Staubli VAL3: feedbackStatus.pgx

public program feedbackStatus(num x_nOutConnFlag)
begin

  // update connection status on port 11002 (feedback server)

  gotoxy(scMonitor, 0,1)
  // 11 characteres: gotoxy(12,1) to insert status
  put(scMonitor, "Port 11002:")
  gotoxy(scMonitor, 12,1)
  switch x_nOutConnFlag
    case -1
      put(scMonitor, "connection lost")
    break
    case 0
      put(scMonitor, "not connected")
    break
    case 1
      put(scMonitor, "connected")
    break
    default
      put(scMonitor, "not connected")
    break
  endSwitch

end
